// TIA Portal V17 export
// export: Created 2024-08-09T12:53:14.1360106Z, ExportSetting WithDefaults, DisplayName Totally Integrated Automation Portal, DisplayVersion V17 Update 7, DisplayName TIA Portal Openness, DisplayVersion V17 Update 7, DisplayName TIA Portal Version Control Interface, DisplayVersion V17, DisplayName STEP 7 Professional, DisplayVersion V17 Update 7, DisplayName STEP 7 Safety, DisplayVersion V17 Update 6, DisplayName WinCC Professional, DisplayVersion V17 Update 7
VAR_GLOBAL   // PLC tag table "LIQUIDE MELANGEUSE"
END_VAR
VAR_GLOBAL CONSTANT   // user constants
   NIV_LIQ_DEBUT_LOT : USInt := 1;
   NIV_LIQ_FIN_CONTROLES : USInt := 10;
   NIV_LIQ_INJ_ENC : USInt := 20;
   NIV_LIQ_CONS_ATTEINTE : USInt := 35;
   NIV_LIQ_FIN_INJ : USInt := 40;
   NIV_LIQ_ATT_FIN_MEL : USInt := 50;
   NIV_LIQ_FIN_LOT : USInt := 255;
END_VAR
